FUNCTION_BLOCK "fbArchiveSlotShipping"
{ S7_Optimized_Access := 'TRUE' }
VERSION : 0.8
   VAR
      slotShipping : Array[1..2] of Struct
         slot : Array[1..1] of "tSlot";
      END_STRUCT;
   END_VAR


BEGIN
END_FUNCTION_BLOCK

